(* Logix 5000 project; controller Corte Emulate 5570 rev 30.12; software revision 30.00 *)

TASK MainTask (continuous, watchdog 500 ms) : MainProgram

MODULES
   Local : Emulate 5570 (ICP 2, rev 30.12)
END_MODULES

PROGRAM MainProgram   (* main routine MainRoutine *)
VAR
   Action_000 : SFC_ACTION := (Status := 16#0020_0000, PauseTimer := 1);
   Action_001 : SFC_ACTION := (Status := 16#0020_0000, PauseTimer := 1);
   Action_002 : SFC_ACTION := (Status := 16#0020_0000, PauseTimer := 1);
   Action_003 : SFC_ACTION := (Status := 16#0020_0000, PauseTimer := 1);
   Action_004 : SFC_ACTION := (Status := 16#0020_0000, PauseTimer := 1);
   Action_005 : SFC_ACTION := (Status := 16#0020_0000, PauseTimer := 1);
   Action_006 : SFC_ACTION := (Status := 16#0020_0000, PauseTimer := 1);
   Action_007 : SFC_ACTION := (Status := 16#0020_0000, PauseTimer := 1);
   Action_008 : SFC_ACTION := (Status := 16#0020_0000, PauseTimer := 1);
   Action_009 : SFC_ACTION := (Status := 16#0020_0000, PauseTimer := 1);
   Action_010 : SFC_ACTION := (Status := 16#0020_0000, PauseTimer := 1);
   Action_011 : SFC_ACTION := (Status := 16#0020_0000, PauseTimer := 1);
   Action_012 : SFC_ACTION := (Status := 16#0020_0000, PauseTimer := 1);
   Action_013 : SFC_ACTION := (Status := 16#0020_0000, PauseTimer := 1);
   Action_014 : SFC_ACTION := (Status := 16#0020_0000, PauseTimer := 1);
   Action_015 : SFC_ACTION := (Status := 16#0020_0000, PauseTimer := 1);
   Action_016 : SFC_ACTION := (Status := 16#0020_0000, PauseTimer := 1);
   Action_017 : SFC_ACTION := (Status := 16#0020_0000, PauseTimer := 1);
   Action_018 : SFC_ACTION := (Status := 16#0020_0000, PauseTimer := 1);
   Action_019 : SFC_ACTION := (Status := 16#0020_0000, PauseTimer := 1);
   Action_020 : SFC_ACTION := (Status := 16#0020_0000, PauseTimer := 1);
   Action_021 : SFC_ACTION := (Status := 16#0020_0000, PauseTimer := 1);
   Action_022 : SFC_ACTION := (Status := 16#0020_0000, PauseTimer := 1);
   Action_023 : SFC_ACTION := (Status := 16#0020_0000, PauseTimer := 1);
   Action_024 : SFC_ACTION := (Status := 16#0020_0000, PauseTimer := 1);
   Action_025 : SFC_ACTION := (Status := 16#0020_0000, PauseTimer := 1);
   Action_026 : SFC_ACTION := (Status := 16#0020_0000, PauseTimer := 1);
   Action_027 : SFC_ACTION := (Status := 16#0020_0000, PauseTimer := 1);
   Action_028 : SFC_ACTION := (Status := 16#0020_0000, PauseTimer := 1);
   Action_029 : SFC_ACTION := (Status := 16#0020_0000, PauseTimer := 1);
   Action_030 : SFC_ACTION := (Status := 16#0020_0000, PauseTimer := 1);
   Action_031 : SFC_ACTION := (Status := 16#0020_0000, PauseTimer := 1);
   Action_032 : SFC_ACTION := (Status := 16#0020_0000, PauseTimer := 1);
   Action_033 : SFC_ACTION := (Status := 16#0020_0000, PauseTimer := 1);
   Action_034 : SFC_ACTION := (Status := 16#0020_0000, PauseTimer := 1);
   Action_035 : SFC_ACTION := (Status := 16#0020_0000, PauseTimer := 1);
   Action_036 : SFC_ACTION := (Status := 16#0020_0000, PauseTimer := 1);
   Counter1 : INT;
   Counter2 : INT;
   H1 : BOOL;
   H2 : BOOL;
   H3 : BOOL;
   L1 : BOOL;
   L10 : BOOL;
   L11 : BOOL;
   L12 : BOOL;
   L2 : BOOL;
   L3 : BOOL;
   L4 : BOOL;
   L5 : BOOL;
   L6 : BOOL;
   L7 : BOOL;
   L8 : BOOL;
   L9 : BOOL;
   MOTOR : BOOL;
   S1 : BOOL;
   S2 : BOOL;
   S3 : BOOL;
   S4 : BOOL;
   S5 : BOOL;
   S6 : BOOL;
   START : BOOL;
   Step_000 : SFC_STEP := (Status := 16#0020_0000, PauseTimer := 1);
   Step_001 : SFC_STEP := (Status := 16#0020_0000, PauseTimer := 1);
   Step_002 : SFC_STEP := (Status := 16#0020_0000, PauseTimer := 1);
   Step_003 : SFC_STEP := (Status := 16#0020_0000, PauseTimer := 1, PRE := 1000);
   Step_004 : SFC_STEP := (Status := 16#0020_0000, PauseTimer := 1);
   Step_005 : SFC_STEP := (Status := 16#0020_0000, PauseTimer := 1);
   Step_006 : SFC_STEP := (Status := 16#0020_0000, PauseTimer := 1);
   Step_007 : SFC_STEP := (Status := 16#0020_0000, PauseTimer := 1);
   Step_008 : SFC_STEP := (Status := 16#0020_0000, PauseTimer := 1);
   Step_009 : SFC_STEP := (Status := 16#0020_0000, PauseTimer := 1);
   Step_010 : SFC_STEP := (Status := 16#0020_0000, PauseTimer := 1);
   Step_011 : SFC_STEP := (Status := 16#0020_0000, PauseTimer := 1);
   Step_012 : SFC_STEP := (Status := 16#0020_0000, PauseTimer := 1);
   Step_013 : SFC_STEP := (Status := 16#0020_0000, PauseTimer := 1);
   Step_014 : SFC_STEP := (Status := 16#0020_0000, PauseTimer := 1);
   Step_015 : SFC_STEP := (Status := 16#0020_0000, PauseTimer := 1);
   Step_016 : SFC_STEP := (Status := 16#0020_0000, PauseTimer := 1);
   Step_017 : SFC_STEP := (Status := 16#0020_0000, PauseTimer := 1);
   Step_018 : SFC_STEP := (Status := 16#0020_0000, PauseTimer := 1);
   Step_019 : SFC_STEP := (Status := 16#0020_0000, PauseTimer := 1, PRE := 1000);
   Step_020 : SFC_STEP := (Status := 16#0020_0000, PauseTimer := 1);
   Step_021 : SFC_STEP := (Status := 16#0020_0000, PauseTimer := 1);
   Step_022 : SFC_STEP := (Status := 16#0020_0000, PauseTimer := 1);
   Step_023 : SFC_STEP := (Status := 16#0020_0000, PauseTimer := 1);
   Step_024 : SFC_STEP := (Status := 16#0020_0000, PauseTimer := 1);
   Step_025 : SFC_STEP := (Status := 16#0020_0000, PauseTimer := 1);
   Step_026 : SFC_STEP := (Status := 16#0020_0000, PauseTimer := 1);
   Step_027 : SFC_STEP := (Status := 16#0020_0000, PauseTimer := 1);
   Step_028 : SFC_STEP := (Status := 16#0020_0000, PauseTimer := 1);
   Step_029 : SFC_STEP := (Status := 16#0020_0000, PauseTimer := 1);
   Step_030 : SFC_STEP := (Status := 16#0020_0000, PauseTimer := 1);
   Step_031 : SFC_STEP := (Status := 16#0020_0000, PauseTimer := 1);
   Step_032 : SFC_STEP := (Status := 16#0020_0000, PauseTimer := 1);
   Step_033 : SFC_STEP := (Status := 16#0020_0000, PauseTimer := 1);
   Step_034 : SFC_STEP := (Status := 16#0020_0000, PauseTimer := 1);
   Step_035 : SFC_STEP := (Status := 16#0020_0000, PauseTimer := 1);
   Step_036 : SFC_STEP := (Status := 16#0020_0000, PauseTimer := 1);
   Tran_000 : BOOL;
   Tran_001 : BOOL;
   Tran_002 : BOOL;
   Tran_003 : BOOL;
   Tran_004 : BOOL;
   Tran_005 : BOOL;
   Tran_006 : BOOL;
   Tran_007 : BOOL;
   Tran_008 : BOOL;
   Tran_009 : BOOL;
   Tran_010 : BOOL;
   Tran_011 : BOOL;
   Tran_012 : BOOL;
   Tran_013 : BOOL;
   Tran_014 : BOOL;
   Tran_015 : BOOL;
   Tran_016 : BOOL;
   Tran_017 : BOOL;
   Tran_018 : BOOL;
   Tran_019 : BOOL;
   Tran_020 : BOOL;
   Tran_021 : BOOL;
   Tran_022 : BOOL;
   Tran_023 : BOOL;
   Tran_024 : BOOL;
   Tran_025 : BOOL;
   Tran_026 : BOOL;
   Tran_027 : BOOL;
   Tran_028 : BOOL;
   Tran_029 : BOOL;
   Tran_030 : BOOL;
   Tran_031 : BOOL;
   Tran_032 : BOOL;
   Tran_033 : BOOL;
   Tran_034 : BOOL;
   Tran_035 : BOOL;
   Tran_036 : BOOL;
   Tran_037 : BOOL;
   Tran_038 : BOOL;
   Tran_039 : BOOL;
   Tran_040 : BOOL;
   Tran_041 : BOOL;
   Tran_042 : BOOL;
   Tran_043 : BOOL;
   Tran_044 : BOOL;
   Tran_045 : BOOL;
   Tran_046 : BOOL;
   Tran_047 : BOOL;
   Tran_048 : BOOL;
   Tran_049 : BOOL;
   Tran_050 : BOOL;
   Tran_051 : BOOL;
   Tran_052 : BOOL;
   Tran_053 : BOOL;
   Tran_054 : BOOL;
   Tran_055 : BOOL;
   Tran_056 : BOOL;
   Tran_057 : BOOL;
   Tran_058 : BOOL;
   Tran_059 : BOOL;
   Y1 : BOOL;
   Y2 : BOOL;
   Y3 : BOOL;
   Y4 : BOOL;
   Y5 : BOOL;
   Y6 : BOOL;
END_VAR

ROUTINE MainRoutine   (* ladder *)
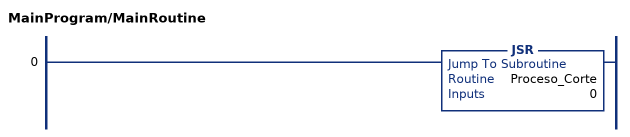
   0: JSR(Proceso_Corte,0);
END_ROUTINE

ROUTINE Proceso_Corte   (* sequential function chart *)
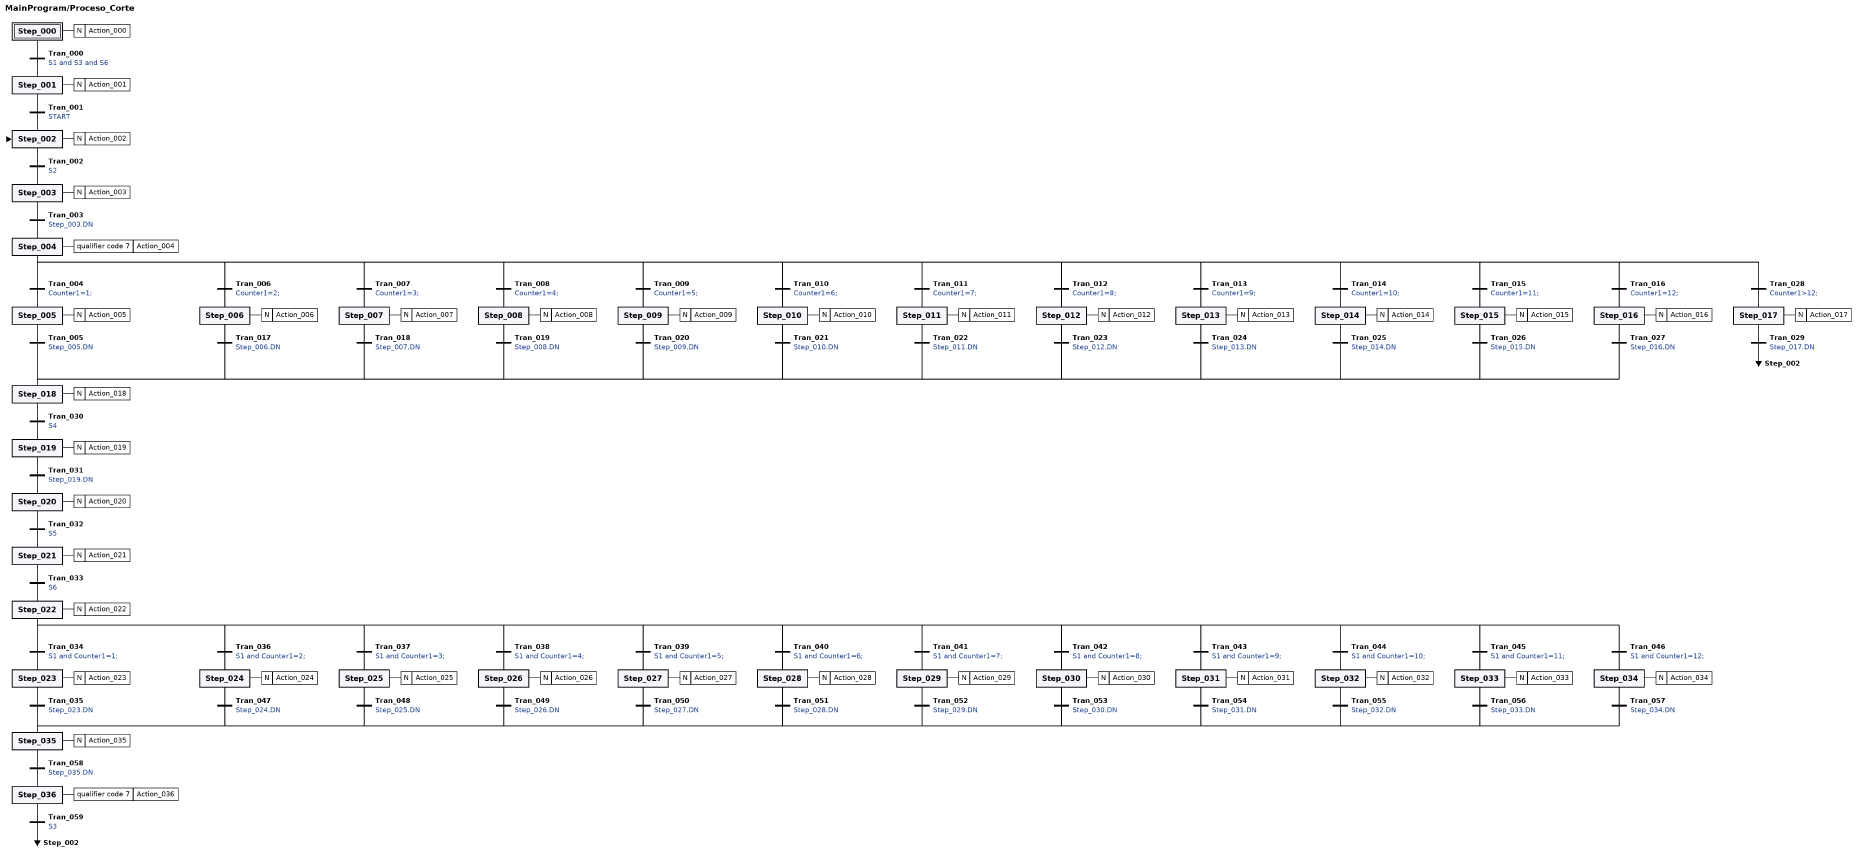
   INITIAL_STEP Step_000:
      ACTION Action_000 (N):
         Y1:=0; Y2:=1; Y3:=0; Y4:=1; Y5:=1; Y6:=0;
         L1:=0; L2:=0; L3:=0; L4:=0; L5:=0; L6:=0;
         L7:=0; L8:=0; L9:=0; L10:=0; L11:=0; L12:=0;
         H1:=0; H2:=0; H3:=0; MOTOR:=0;
         Counter1:=0; Counter2:=0;
         
         
         
         
      END_ACTION
   END_STEP
   TRANSITION Tran_000 FROM Step_000 TO Step_001
      := S1 and S3 and S6
   END_TRANSITION
   STEP Step_001:
      ACTION Action_001 (N):
         H1:=1; H2:=0; H3:=0;
         Y2:=0; Y4:=0; Y5:=0;
      END_ACTION
   END_STEP
   TRANSITION Tran_001 FROM Step_001 TO Step_002
      := START
   END_TRANSITION
   STEP Step_002:
      ACTION Action_002 (N):
         Y1:=1;
         MOTOR:=1;
         H2:=1;
         H1:=0;
      END_ACTION
   END_STEP
   TRANSITION Tran_002 FROM Step_002 TO Step_003
      := S2
   END_TRANSITION
   STEP Step_003:
      ACTION Action_003 (N):
         Y1:=0;
      END_ACTION
   END_STEP
   TRANSITION Tran_003 FROM Step_003 TO Step_004
      := Step_003.DN
   END_TRANSITION
   STEP Step_004:
      ACTION Action_004 (qualifier code 7):
         Counter1:=Counter1+1;
      END_ACTION
   END_STEP
   TRANSITION Tran_004 FROM Step_004 TO Step_005
      := Counter1=1;
   END_TRANSITION
   TRANSITION Tran_006 FROM Step_004 TO Step_006
      := Counter1=2;
   END_TRANSITION
   TRANSITION Tran_007 FROM Step_004 TO Step_007
      := Counter1=3;
   END_TRANSITION
   TRANSITION Tran_008 FROM Step_004 TO Step_008
      := Counter1=4;
   END_TRANSITION
   TRANSITION Tran_009 FROM Step_004 TO Step_009
      := Counter1=5;
   END_TRANSITION
   TRANSITION Tran_010 FROM Step_004 TO Step_010
      := Counter1=6;
   END_TRANSITION
   TRANSITION Tran_011 FROM Step_004 TO Step_011
      := Counter1=7;
   END_TRANSITION
   TRANSITION Tran_012 FROM Step_004 TO Step_012
      := Counter1=8;
   END_TRANSITION
   TRANSITION Tran_013 FROM Step_004 TO Step_013
      := Counter1=9;
   END_TRANSITION
   TRANSITION Tran_014 FROM Step_004 TO Step_014
      := Counter1=10;
   END_TRANSITION
   TRANSITION Tran_015 FROM Step_004 TO Step_015
      := Counter1=11;
   END_TRANSITION
   TRANSITION Tran_016 FROM Step_004 TO Step_016
      := Counter1=12;
   END_TRANSITION
   TRANSITION Tran_028 FROM Step_004 TO Step_017
      := Counter1>12;
   END_TRANSITION
   STEP Step_005:
      ACTION Action_005 (N):
         L1:=1;
         
      END_ACTION
   END_STEP
   STEP Step_006:
      ACTION Action_006 (N):
         L2:=1;
         
      END_ACTION
   END_STEP
   STEP Step_007:
      ACTION Action_007 (N):
         L3:=1;
         
         
      END_ACTION
   END_STEP
   STEP Step_008:
      ACTION Action_008 (N):
         L4:=1;
         
      END_ACTION
   END_STEP
   STEP Step_009:
      ACTION Action_009 (N):
         L5:=1;
         
      END_ACTION
   END_STEP
   STEP Step_010:
      ACTION Action_010 (N):
         L6:=1;
         
      END_ACTION
   END_STEP
   STEP Step_011:
      ACTION Action_011 (N):
         L7:=1;
         
      END_ACTION
   END_STEP
   STEP Step_012:
      ACTION Action_012 (N):
         L8:=1;
         
      END_ACTION
   END_STEP
   STEP Step_013:
      ACTION Action_013 (N):
         L9:=1;
         
      END_ACTION
   END_STEP
   STEP Step_014:
      ACTION Action_014 (N):
         L10:=1;
         
      END_ACTION
   END_STEP
   STEP Step_015:
      ACTION Action_015 (N):
         L11:=1;
         
      END_ACTION
   END_STEP
   STEP Step_016:
      ACTION Action_016 (N):
         L12:=1;
         
      END_ACTION
   END_STEP
   STEP Step_017:
      ACTION Action_017 (N):
         Counter1:=0;
         
      END_ACTION
   END_STEP
   TRANSITION Tran_005 FROM Step_005 TO Step_018
      := Step_005.DN
   END_TRANSITION
   TRANSITION Tran_017 FROM Step_006 TO Step_018
      := Step_006.DN
   END_TRANSITION
   TRANSITION Tran_018 FROM Step_007 TO Step_018
      := Step_007.DN
   END_TRANSITION
   TRANSITION Tran_019 FROM Step_008 TO Step_018
      := Step_008.DN
   END_TRANSITION
   TRANSITION Tran_020 FROM Step_009 TO Step_018
      := Step_009.DN
   END_TRANSITION
   TRANSITION Tran_021 FROM Step_010 TO Step_018
      := Step_010.DN
   END_TRANSITION
   TRANSITION Tran_022 FROM Step_011 TO Step_018
      := Step_011.DN
   END_TRANSITION
   TRANSITION Tran_023 FROM Step_012 TO Step_018
      := Step_012.DN
   END_TRANSITION
   TRANSITION Tran_024 FROM Step_013 TO Step_018
      := Step_013.DN
   END_TRANSITION
   TRANSITION Tran_025 FROM Step_014 TO Step_018
      := Step_014.DN
   END_TRANSITION
   TRANSITION Tran_026 FROM Step_015 TO Step_018
      := Step_015.DN
   END_TRANSITION
   TRANSITION Tran_027 FROM Step_016 TO Step_018
      := Step_016.DN
   END_TRANSITION
   TRANSITION Tran_029 FROM Step_017 TO Step_002
      := Step_017.DN
   END_TRANSITION
   STEP Step_018:
      ACTION Action_018 (N):
         Y3:=1;
      END_ACTION
   END_STEP
   TRANSITION Tran_030 FROM Step_018 TO Step_019
      := S4
   END_TRANSITION
   STEP Step_019:
      ACTION Action_019 (N):
         Y3:=0;
      END_ACTION
   END_STEP
   TRANSITION Tran_031 FROM Step_019 TO Step_020
      := Step_019.DN
   END_TRANSITION
   STEP Step_020:
      ACTION Action_020 (N):
         Y6:=1;
      END_ACTION
   END_STEP
   TRANSITION Tran_032 FROM Step_020 TO Step_021
      := S5
   END_TRANSITION
   STEP Step_021:
      ACTION Action_021 (N):
         Y5:=1;
         Y6:=0;
      END_ACTION
   END_STEP
   TRANSITION Tran_033 FROM Step_021 TO Step_022
      := S6
   END_TRANSITION
   STEP Step_022:
      ACTION Action_022 (N):
         Y2:=1;
         Y5:=0;
      END_ACTION
   END_STEP
   TRANSITION Tran_034 FROM Step_022 TO Step_023
      := S1 and Counter1=1;
   END_TRANSITION
   TRANSITION Tran_036 FROM Step_022 TO Step_024
      := S1 and Counter1=2;
   END_TRANSITION
   TRANSITION Tran_037 FROM Step_022 TO Step_025
      := S1 and Counter1=3;
   END_TRANSITION
   TRANSITION Tran_038 FROM Step_022 TO Step_026
      := S1 and Counter1=4;
   END_TRANSITION
   TRANSITION Tran_039 FROM Step_022 TO Step_027
      := S1 and Counter1=5;
   END_TRANSITION
   TRANSITION Tran_040 FROM Step_022 TO Step_028
      := S1 and Counter1=6;
   END_TRANSITION
   TRANSITION Tran_041 FROM Step_022 TO Step_029
      := S1 and Counter1=7;
   END_TRANSITION
   TRANSITION Tran_042 FROM Step_022 TO Step_030
      := S1 and Counter1=8;
   END_TRANSITION
   TRANSITION Tran_043 FROM Step_022 TO Step_031
      := S1 and Counter1=9;
   END_TRANSITION
   TRANSITION Tran_044 FROM Step_022 TO Step_032
      := S1 and Counter1=10;
   END_TRANSITION
   TRANSITION Tran_045 FROM Step_022 TO Step_033
      := S1 and Counter1=11;
   END_TRANSITION
   TRANSITION Tran_046 FROM Step_022 TO Step_034
      := S1 and Counter1=12;
   END_TRANSITION
   STEP Step_023:
      ACTION Action_023 (N):
         L1:=0;
         
      END_ACTION
   END_STEP
   STEP Step_024:
      ACTION Action_024 (N):
         L2:=0;
         
      END_ACTION
   END_STEP
   STEP Step_025:
      ACTION Action_025 (N):
         L3:=0;
         
         
      END_ACTION
   END_STEP
   STEP Step_026:
      ACTION Action_026 (N):
         L4:=0;
         
      END_ACTION
   END_STEP
   STEP Step_027:
      ACTION Action_027 (N):
         L5:=0;
         
      END_ACTION
   END_STEP
   STEP Step_028:
      ACTION Action_028 (N):
         L6:=0;
         
      END_ACTION
   END_STEP
   STEP Step_029:
      ACTION Action_029 (N):
         L7:=0;
         
      END_ACTION
   END_STEP
   STEP Step_030:
      ACTION Action_030 (N):
         L8:=0;
         
      END_ACTION
   END_STEP
   STEP Step_031:
      ACTION Action_031 (N):
         L9:=0;
         
      END_ACTION
   END_STEP
   STEP Step_032:
      ACTION Action_032 (N):
         L10:=0;
         
      END_ACTION
   END_STEP
   STEP Step_033:
      ACTION Action_033 (N):
         L11:=0;
         
      END_ACTION
   END_STEP
   STEP Step_034:
      ACTION Action_034 (N):
         L12:=0;
         
      END_ACTION
   END_STEP
   TRANSITION Tran_035 FROM Step_023 TO Step_035
      := Step_023.DN
   END_TRANSITION
   TRANSITION Tran_047 FROM Step_024 TO Step_035
      := Step_024.DN
   END_TRANSITION
   TRANSITION Tran_048 FROM Step_025 TO Step_035
      := Step_025.DN
   END_TRANSITION
   TRANSITION Tran_049 FROM Step_026 TO Step_035
      := Step_026.DN
   END_TRANSITION
   TRANSITION Tran_050 FROM Step_027 TO Step_035
      := Step_027.DN
   END_TRANSITION
   TRANSITION Tran_051 FROM Step_028 TO Step_035
      := Step_028.DN
   END_TRANSITION
   TRANSITION Tran_052 FROM Step_029 TO Step_035
      := Step_029.DN
   END_TRANSITION
   TRANSITION Tran_053 FROM Step_030 TO Step_035
      := Step_030.DN
   END_TRANSITION
   TRANSITION Tran_054 FROM Step_031 TO Step_035
      := Step_031.DN
   END_TRANSITION
   TRANSITION Tran_055 FROM Step_032 TO Step_035
      := Step_032.DN
   END_TRANSITION
   TRANSITION Tran_056 FROM Step_033 TO Step_035
      := Step_033.DN
   END_TRANSITION
   TRANSITION Tran_057 FROM Step_034 TO Step_035
      := Step_034.DN
   END_TRANSITION
   STEP Step_035:
      ACTION Action_035 (N):
         Y4:=1;
         Y2:=0;
      END_ACTION
   END_STEP
   TRANSITION Tran_058 FROM Step_035 TO Step_036
      := Step_035.DN
   END_TRANSITION
   STEP Step_036:
      ACTION Action_036 (qualifier code 7):
         Counter2:=Counter2+1;
      END_ACTION
   END_STEP
   TRANSITION Tran_059 FROM Step_036 TO Step_002
      := S3
   END_TRANSITION
END_ROUTINE
END_PROGRAM
